{attribute 'linkalways'} 
{attribute 'no_explicit_call' := 'This FB is a CLASS and must be accessed using methods or properties'}
{attribute 'enable_dynamic_creation'}
FUNCTION_BLOCK Mc2Axis IMPLEMENTS Axis
VAR
	axis_ref : Tc2_Mc2.Axis_Ref;
	power_fb : Tc2_Mc2.Mc_Power;
	reset_fb : Tc2_Mc2.Mc_Reset;
	halt_fb : Tc2_Mc2.Mc_Halt;
	stop_fb : Tc2_Mc2.Mc_Stop;
END_VAR

METHOD PUBLIC CyclicCall
power_fb(Axis := axis_ref);
reset_fb(Axis := axis_ref);
halt_fb(Axis := axis_ref);
stop_fb(Axis := axis_ref);
axis_ref.ReadStatus();
END_METHOD

METHOD PUBLIC Disable
power_fb.Enable := FALSE;
power_fb.Enable_Positive := FALSE;
power_fb.Enable_Negative := FALSE;
END_METHOD

METHOD PUBLIC DisableNegative
power_fb.Enable_Negative := FALSE;
END_METHOD

METHOD PUBLIC DisablePositive
power_fb.Enable_Positive := FALSE;
END_METHOD

METHOD PUBLIC Enable
power_fb.Enable := TRUE;
END_METHOD

METHOD PUBLIC EnableNegative
power_fb.Enable_Negative := TRUE;
END_METHOD

METHOD PUBLIC EnablePositive
power_fb.Enable_Positive := TRUE;
END_METHOD

{attribute 'monitoring' := 'call'}
PROPERTY PUBLIC ErrorId : UDINT
GET // PUBLIC
ErrorId := axis_ref.Status.ErrorId;
END_GET
END_PROPERTY

METHOD PUBLIC GearIn : AsyncCommand
VAR_INPUT
	master_axis : Axis;
	numerator : LREAL;
	denominator : UINT := 1;
	//acceleration : LREAL := 0;
	//deceleration : LREAL := 0;
	//jerk : LREAL := 0;
	//buffer_mode	: MotionBufferMode := MotionBufferMode.Aborting;
END_VAR
VAR
	mc2_master_axis : POINTER TO Mc2Axis;
	command_pointer : POINTER TO GearInCommand;
END_VAR
IF __QUERYPOINTER(master_axis, mc2_master_axis) THEN
	command_pointer := __NEW(
		GearInCommand(
			master_axis := mc2_master_axis^,
			slave_axis := THIS^,
			numerator := numerator,
			denominator := denominator
		)
	);
	
	GearIn := command_pointer^;
END_IF
END_METHOD

METHOD PUBLIC GearOut : AsyncCommand
VAR
	command_pointer : POINTER TO GearOutCommand;
END_VAR
command_pointer := __NEW(
	GearOutCommand(
		axis := THIS^
	)
);

GearOut := command_pointer^;
END_METHOD

METHOD PUBLIC Halt : MoveCommand
VAR_INPUT
	deceleration : LREAL := 0;
	jerk : LREAL := 0;
	buffer_mode	: MotionBufferMode := MotionBufferMode.Aborting;
END_VAR
VAR
	command_pointer : POINTER TO HaltCommand;
END_VAR
command_pointer := __NEW(
	HaltCommand(
		axis := THIS^,
		deceleration := deceleration,
		jerk := jerk,
		buffer_mode := buffer_mode
	)
);

Halt := command_pointer^;
END_METHOD

{attribute 'monitoring' := 'call'}
PROPERTY PUBLIC HasBeenStopped : BOOL
GET // PUBLIC
HasBeenStopped := axis_ref.Status.HasBeenStopped;
END_GET
END_PROPERTY

{attribute 'monitoring' := 'call'}
PROPERTY PUBLIC HasJob : BOOL
GET // PUBLIC
HasJob := axis_ref.Status.HasJob;
END_GET
END_PROPERTY

{attribute 'monitoring' := 'call'}
PROPERTY PUBLIC IsAccelerating : BOOL
GET // PUBLIC
IsAccelerating := axis_ref.Status.Accelerating;
END_GET
END_PROPERTY

{attribute 'monitoring' := 'call'}
PROPERTY PUBLIC IsBusyHoming : BOOL
GET // PUBLIC
IsBusyHoming := axis_ref.Status.HomingBusy;
END_GET
END_PROPERTY

{attribute 'monitoring' := 'call'}
PROPERTY PUBLIC IsCamDataQueued : BOOL
GET // PUBLIC
IsCamDataQueued := axis_ref.Status.CamDataQueued;
END_GET
END_PROPERTY

{attribute 'monitoring' := 'call'}
PROPERTY PUBLIC IsCamScalingPending : BOOL
GET // PUBLIC
IsCamScalingPending := axis_ref.Status.CamScalingPending;
END_GET
END_PROPERTY

{attribute 'monitoring' := 'call'}
PROPERTY PUBLIC IsCamTableQueued : BOOL
GET // PUBLIC
IsCamTableQueued := axis_ref.Status.CamTableQueued;
END_GET
END_PROPERTY

{attribute 'monitoring' := 'call'}
 PROPERTY PUBLIC IsCommandBuffered : BOOL
GET // PUBLIC
IsCommandBuffered := axis_ref.Status.CmdBuffered;
END_GET
END_PROPERTY

{attribute 'monitoring' := 'call'}
PROPERTY PUBLIC IsCompensating : BOOL
GET // PUBLIC
IsCompensating := axis_ref.Status.Compensating;
END_GET
END_PROPERTY

{attribute 'monitoring' := 'call'}
PROPERTY PUBLIC IsConstantVelocity : BOOL
GET // PUBLIC
IsConstantVelocity := axis_ref.Status.ConstantVelocity;
END_GET
END_PROPERTY

{attribute 'monitoring' := 'call'}
PROPERTY PUBLIC IsContinuousMotion : BOOL
GET // PUBLIC
IsContinuousMotion := axis_ref.Status.ContinuousMotion;
END_GET
END_PROPERTY

{attribute 'monitoring' := 'call'}
PROPERTY PUBLIC IsControlLoopClosed : BOOL
GET // PUBLIC
IsControlLoopClosed := axis_ref.Status.ControlLoopClosed;
END_GET
END_PROPERTY

{attribute 'monitoring' := 'call'}
PROPERTY PUBLIC IsCoupled : BOOL
GET // PUBLIC
IsCoupled := axis_ref.Status.Coupled;
END_GET
END_PROPERTY

{attribute 'monitoring' := 'call'}
PROPERTY PUBLIC IsDecelerating : BOOL
GET // PUBLIC
IsDecelerating := axis_ref.Status.Decelerating;
END_GET
END_PROPERTY

{attribute 'monitoring' := 'call'}
PROPERTY PUBLIC IsDisabled : BOOL
GET // PUBLIC
IsDisabled := axis_ref.Status.Disabled;
END_GET
END_PROPERTY

{attribute 'monitoring' := 'call'}
PROPERTY PUBLIC IsDiscreteMotion : BOOL
GET // PUBLIC
END_GET
END_PROPERTY

{attribute 'monitoring' := 'call'}
PROPERTY PUBLIC IsDriveDeviceErrored : BOOL
GET // PUBLIC
IsDriveDeviceErrored := axis_ref.Status.Error;
END_GET
END_PROPERTY

{attribute 'monitoring' := 'call'}
PROPERTY PUBLIC IsErrored : BOOL
GET // PUBLIC
IsErrored := axis_ref.Status.Error;
END_GET
END_PROPERTY

{attribute 'monitoring' := 'call'}
PROPERTY PUBLIC IsErrorStop : BOOL
GET // PUBLIC
IsErrorStop := axis_ref.Status.ErrorStop;
END_GET
END_PROPERTY

{attribute 'monitoring' := 'call'}
PROPERTY PUBLIC IsExternalLatchValid : BOOL
GET // PUBLIC
IsExternalLatchValid := axis_ref.Status.ExternalLatchValid;
END_GET
END_PROPERTY

{attribute 'monitoring' := 'call'}
PROPERTY PUBLIC IsExtSetPointGenEnabled : BOOL
GET // PUBLIC
IsExtSetPointGenEnabled := axis_ref.Status.ExtSetPointGenEnabled;
END_GET
END_PROPERTY

{attribute 'monitoring' := 'call'}
PROPERTY PUBLIC IsHomed : BOOL
GET // PUBLIC
IsHomed := axis_ref.Status.Homed;
END_GET
END_PROPERTY

{attribute 'monitoring' := 'call'}
PROPERTY PUBLIC IsHoming : BOOL
GET // PUBLIC
IsHoming := axis_ref.Status.Homing;
END_GET
END_PROPERTY

{attribute 'monitoring' := 'call'}
PROPERTY PUBLIC IsInPositionArea : BOOL
GET // PUBLIC
IsInPositionArea := axis_ref.Status.InPositionArea;
END_GET
END_PROPERTY

{attribute 'monitoring' := 'call'}
PROPERTY PUBLIC IsInTargetPosition : BOOL
GET // PUBLIC
IsInTargetPosition := axis_ref.Status.InTargetPosition;
END_GET
END_PROPERTY

{attribute 'monitoring' := 'call'}
PROPERTY PUBLIC IsIoDataInvalid : BOOL
GET // PUBLIC
IsIoDataInvalid := axis_ref.Status.IoDataInvalid;
END_GET
END_PROPERTY

{attribute 'monitoring' := 'call'}
PROPERTY PUBLIC IsMotionCommandsLocked : BOOL
GET // PUBLIC
IsMotionCommandsLocked := axis_ref.Status.MotionCommandsLocked;
END_GET
END_PROPERTY

{attribute 'monitoring' := 'call'}
PROPERTY PUBLIC IsMoving : BOOL
GET // PUBLIC
IsMoving := axis_ref.Status.Moving;
END_GET
END_PROPERTY

{attribute 'monitoring' := 'call'}
PROPERTY PUBLIC IsNegativeDirection : BOOL
GET // PUBLIC
IsNegativeDirection := axis_ref.Status.NegativeDirection;
END_GET
END_PROPERTY

{attribute 'monitoring' := 'call'}
PROPERTY PUBLIC IsNewTargetPosition : BOOL
GET // PUBLIC
IsNewTargetPosition := axis_ref.Status.NewTargetPosition;
END_GET
END_PROPERTY

{attribute 'monitoring' := 'call'}
PROPERTY PUBLIC IsNotMoving : BOOL
GET // PUBLIC
IsNotMoving := axis_ref.Status.NotMoving;
END_GET
END_PROPERTY

{attribute 'monitoring' := 'call'}
PROPERTY PUBLIC IsOperational : BOOL
GET // PUBLIC
IsOperational := axis_ref.Status.Operational;
END_GET
END_PROPERTY

{attribute 'monitoring' := 'call'}
PROPERTY PUBLIC IsPointToPointMode : BOOL
GET // PUBLIC
IsPointToPointMode := axis_ref.Status.PTPmode;
END_GET
END_PROPERTY

{attribute 'monitoring' := 'call'}
PROPERTY PUBLIC IsPositiveDirection : BOOL
GET // PUBLIC
IsPositiveDirection := axis_ref.Status.PositiveDirection;
END_GET
END_PROPERTY

{attribute 'monitoring' := 'call'}
PROPERTY PUBLIC IsProtected : BOOL
GET // PUBLIC
IsProtected := axis_ref.Status.ProtectedMode;
END_GET
END_PROPERTY

{attribute 'monitoring' := 'call'}
PROPERTY PUBLIC IsSoftLimitMaxExceeded : BOOL
GET // PUBLIC
IsSoftLimitMaxExceeded := axis_ref.Status.SoftLimitMaxExceeded;
END_GET
END_PROPERTY

{attribute 'monitoring' := 'call'}
PROPERTY PUBLIC IsSoftLimitMinExceeded : BOOL
GET // PUBLIC
IsSoftLimitMinExceeded := axis_ref.Status.SoftLimitMinExceeded;
END_GET
END_PROPERTY

{attribute 'monitoring' := 'call'}
PROPERTY PUBLIC IsStandstill : BOOL
GET // PUBLIC
IsStandstill := axis_ref.Status.StandStill;
END_GET
END_PROPERTY

{attribute 'monitoring' := 'call'}
PROPERTY PUBLIC IsStopping : BOOL
GET // PUBLIC
IsStopping := axis_ref.Status.Stopping;
END_GET
END_PROPERTY

{attribute 'monitoring' := 'call'}
PROPERTY PUBLIC IsSynchronisedMotion : BOOL
GET // PUBLIC
IsSynchronisedMotion := axis_ref.Status.SynchronizedMotion;
END_GET
END_PROPERTY

PROPERTY PUBLIC Mc2AxisRef : REFERENCE TO Tc2_Mc2.Axis_Ref
GET // PUBLIC
Mc2AxisRef REF= THIS^.axis_ref;
END_GET
END_PROPERTY

{attribute 'monitoring' := 'call'}
PROPERTY PUBLIC MotionState : AxisMotionState
GET // PUBLIC
CASE axis_ref.Status.MotionState OF
	Tc2_Mc2.Mc_AxisState_Disabled: MotionState := AxisMotionState.Disabled;
	Tc2_Mc2.Mc_AxisState_Standstill: MotionState := AxisMotionState.Standstill;
	Tc2_Mc2.Mc_AxisState_ErrorStop: MotionState := AxisMotionState.ErrorStop;
	Tc2_Mc2.Mc_AxisState_Stopping: MotionState := AxisMotionState.Stopping;
	Tc2_Mc2.Mc_AxisState_Homing: MotionState := AxisMotionState.Homing;
	Tc2_Mc2.Mc_AxisState_DiscreteMotion: MotionState := AxisMotionState.DiscreteMotion;
	Tc2_Mc2.Mc_AxisState_ContinousMotion: MotionState := AxisMotionState.ContinuousMotion;
	Tc2_Mc2.Mc_AxisState_SynchronizedMotion: MotionState := AxisMotionState.SynchronisedMotion;
ELSE
	MotionState := AxisMotionState.Undefined;
END_CASE
END_GET
END_PROPERTY

METHOD PUBLIC MoveAbsolute : MoveCommand
VAR_INPUT
	position : LREAL;
	velocity : LREAL;
	acceleration : LREAL := 0;
	deceleration : LREAL := 0;
	jerk : LREAL := 0;
	buffer_mode	: MotionBufferMode := MotionBufferMode.Aborting;
END_VAR
VAR
	command_pointer : POINTER TO MoveAbsoluteCommand;
END_VAR
command_pointer := __NEW(
	MoveAbsoluteCommand(
		axis := THIS^,
		position := position,
		velocity := velocity,
		acceleration := acceleration,
		deceleration := deceleration,
		jerk := jerk,
		buffer_mode := buffer_mode
	)
);

MoveAbsolute := command_pointer^;
END_METHOD

METHOD PUBLIC MoveContinuousAbsolute : MoveCommand
VAR_INPUT
	position : LREAL;
	velocity : LREAL;
	acceleration : LREAL := 0;
	deceleration : LREAL := 0;
	jerk : LREAL := 0;
	buffer_mode	: MotionBufferMode := MotionBufferMode.Aborting;
END_VAR
VAR
	command_pointer : POINTER TO MoveContinuousAbsoluteCommand;
END_VAR
command_pointer := __NEW(
	MoveContinuousAbsoluteCommand(
		axis := THIS^,
		position := position,
		velocity := velocity,
		acceleration := acceleration,
		deceleration := deceleration,
		jerk := jerk,
		buffer_mode := buffer_mode
	)
);

MoveContinuousAbsolute := command_pointer^;
END_METHOD

METHOD PUBLIC MoveContinuousRelative : MoveCommand
VAR_INPUT
	distance : LREAL;
	velocity : LREAL;
	acceleration : LREAL := 0;
	deceleration : LREAL := 0;
	jerk : LREAL := 0;
	buffer_mode	: MotionBufferMode := MotionBufferMode.Aborting;
END_VAR
VAR
	command_pointer : POINTER TO MoveContinuousRelativeCommand;
END_VAR
command_pointer := __NEW(
	MoveContinuousRelativeCommand(
		axis := THIS^,
		distance := distance,
		velocity := velocity,
		acceleration := acceleration,
		deceleration := deceleration,
		jerk := jerk,
		buffer_mode := buffer_mode
	)
);

MoveContinuousRelative := command_pointer^;
END_METHOD

METHOD PUBLIC MoveModulo : MoveCommand
VAR_INPUT
	position : LREAL;
	direction : MotionDirection;
	velocity : LREAL;
	acceleration : LREAL := 0;
	deceleration : LREAL := 0;
	jerk : LREAL := 0;
	buffer_mode	: MotionBufferMode := MotionBufferMode.Aborting;
END_VAR
VAR
	command_pointer : POINTER TO MoveModuloCommand;
END_VAR
command_pointer := __NEW(
	MoveModuloCommand(
		axis := THIS^,
		position := position,
		direction := direction,
		velocity := velocity,
		acceleration := acceleration,
		deceleration := deceleration,
		jerk := jerk,
		buffer_mode := buffer_mode
	)
);

MoveModulo := command_pointer^;
END_METHOD

METHOD PUBLIC MoveRelative : MoveCommand
VAR_INPUT
	distance : LREAL;
	velocity : LREAL;
	acceleration : LREAL := 0;
	deceleration : LREAL := 0;
	jerk : LREAL := 0;
	buffer_mode	: MotionBufferMode := MotionBufferMode.Aborting;
END_VAR
VAR
	command_pointer : POINTER TO MoveRelativeCommand;
END_VAR
command_pointer := __NEW(
	MoveRelativeCommand(
		axis := THIS^,
		distance := distance,
		velocity := velocity,
		acceleration := acceleration,
		deceleration := deceleration,
		jerk := jerk,
		buffer_mode := buffer_mode
	)
);

MoveRelative := command_pointer^;
END_METHOD

METHOD PUBLIC MoveVelocity : MoveCommand
VAR_INPUT
	velocity : LREAL;
	acceleration : LREAL := 0;
	deceleration : LREAL := 0;
	jerk : LREAL := 0;
	buffer_mode	: MotionBufferMode := MotionBufferMode.Aborting;
END_VAR
VAR
	command_pointer : POINTER TO MoveVelocityCommand;
END_VAR
command_pointer := __NEW(
	MoveVelocityCommand(
		axis := THIS^,
		velocity := velocity,
		acceleration := acceleration,
		deceleration := deceleration,
		jerk := jerk,
		buffer_mode := buffer_mode
	)
);

MoveVelocity := command_pointer^;
END_METHOD

PROPERTY PUBLIC OpMode : Tc2_Mc2.St_AxisOpModes
GET // PUBLIC
OpMode := axis_ref.Status.OpMode;
END_GET
END_PROPERTY

METHOD PUBLIC Stop : MoveCommand
VAR_INPUT
	deceleration : LREAL := 0;
	jerk : LREAL := 0;
END_VAR
VAR
	command_pointer : POINTER TO StopCommand;
END_VAR
command_pointer := __NEW(
	StopCommand(
		axis := THIS^,
		deceleration := deceleration,
		jerk := jerk
	)
);

Stop := command_pointer^;
END_METHOD

END_FUNCTION_BLOCK

(* stored: Version 1.1.0.1
   POU Mc2Axis: Id {f6d24d44-bf88-05ab-17dd-e51bfbadd54a}, SpecialFunc None
   Folder Administrative: Id {c7a39c65-0d79-0e29-1377-7896a907f259}
   Folder Cyclic: Id {4bf04a9e-5f39-0347-2cc3-7f566b01be46}
   Folder Motion: Id {042d880c-d6a7-0bf4-26fc-fbf1514355b4}
   Folder Coupling: Id {c0c3d91b-c064-008c-3bc5-b7d09afefae3}
   Folder PointToPoint: Id {f7c42b14-1338-020f-0e42-fbe1e01f13ed}
   Folder Properties: Id {14bd5cf8-6829-0857-0543-912990d6f17c}
   Folder Error: Id {2ffa55bd-1a34-0c90-1876-f6f0946a309e}
   Folder States: Id {06982f99-509a-0977-0c86-36e4c9e4d884}
   Method CyclicCall: Id {c3d150dc-498f-087b-1e2a-cb28255a9a2e}
   Method Disable: Id {4475c6cd-2c80-0d86-32a6-2a6f85fa4e57}
   Method DisableNegative: Id {ab9e5fd9-cc11-0564-18aa-e34304f4e2e1}
   Method DisablePositive: Id {a7b584fc-cefd-0b94-3aad-fa7d09eaf38c}
   Method Enable: Id {51a4f218-30db-0a36-1b4f-54113e679d4a}
   Method EnableNegative: Id {1b82506a-a2bc-0e96-166c-a270fe33b5e2}
   Method EnablePositive: Id {5bc6496b-cc67-0922-28fc-331c9ad48fe1}
   Property ErrorId: Id {78f66620-fc8b-04ba-2c81-52c0f1fef6cb}
   Get Get: Id {572858b0-3000-039e-294f-09db91a746f0}
   Method GearIn: Id {19d44698-3c91-0578-1b51-8d7bddf03ae4}
   Method GearOut: Id {9f828a07-ad5e-0a29-08a3-d170a741d665}
   Method Halt: Id {bd9a8884-e367-05ac-2011-44121e4bfe1a}
   Property HasBeenStopped: Id {5da5e438-a929-084d-1690-b4c7d430baa3}
   Get Get: Id {05db3da7-bc46-0833-1b83-d37a59337621}
   Property HasJob: Id {523d496b-9657-07d6-055e-41f49b8ff99e}
   Get Get: Id {c3ce1acb-5d1c-0428-06e4-a53819984a3e}
   Property IsAccelerating: Id {ef93bcd0-2e43-098c-1e45-93ea63d85c21}
   Get Get: Id {3748b6f5-bad3-03a0-00b8-5541692d4281}
   Property IsBusyHoming: Id {78e0242c-43f6-00dd-1c0b-3a112bedd1f3}
   Get Get: Id {26cefb18-7e13-0f7c-3fd5-9a2d9a945033}
   Property IsCamDataQueued: Id {bfa5e2c6-a1b8-072e-1343-f2c82e2465be}
   Get Get: Id {0b42bbbc-7152-0758-1356-6a1b6ab20d4c}
   Property IsCamScalingPending: Id {de860177-b0c1-0299-154b-3806a6cdca90}
   Get Get: Id {766aa1a8-0d4f-0a15-39e4-a4660b05a7ae}
   Property IsCamTableQueued: Id {75ed77cd-a788-0e3f-31e7-de98fdd30099}
   Get Get: Id {d7ca3a57-bd1e-0e46-35f4-470c422ef820}
   Property IsCommandBuffered: Id {b037e227-a8b9-0e70-281b-08080b252061}
   Get Get: Id {8a4994b4-3b18-006c-3fb6-5613e0d8d1ee}
   Property IsCompensating: Id {316b11c2-e12a-069f-0be2-e4005b9003d4}
   Get Get: Id {fbc2ddf1-0a8a-0035-3b7a-a7896e19c528}
   Property IsConstantVelocity: Id {6a4d0ff6-a626-0141-307e-e4fe966b6439}
   Get Get: Id {8d2e3362-7b09-0633-0b5c-d5df8abd82b4}
   Property IsContinuousMotion: Id {9f4ef97f-2075-0ac0-350c-4a0af1ec6345}
   Get Get: Id {8ab7cb67-9d1e-0111-03e1-3647dd557e65}
   Property IsControlLoopClosed: Id {486a5c27-9a7c-0132-2b3d-22502f8b0d89}
   Get Get: Id {2062416c-cf8c-08bc-344f-0ef2f454f4b4}
   Property IsCoupled: Id {0e90c18b-5f7e-097f-1af7-f4b40426fa87}
   Get Get: Id {482e08a2-b9fb-0005-3233-477b456b0cbc}
   Property IsDecelerating: Id {5afc1dd6-c5b1-023c-2124-55b5060fb994}
   Get Get: Id {65bd9ee6-64dd-05fd-1de9-d2cfe2928e77}
   Property IsDisabled: Id {f757a26e-d51f-0b87-3f2a-165df82210b7}
   Get Get: Id {360a4cab-ee53-0d36-1188-4ca485d88d9c}
   Property IsDiscreteMotion: Id {6128acf7-fffa-0b89-0bd3-268f2e3ef87f}
   Get Get: Id {a134065a-97d7-092e-1f91-aec42a5fe214}
   Property IsDriveDeviceErrored: Id {8fba9b9f-e00b-0afa-1a40-033c77c15f6d}
   Get Get: Id {530d8c63-b6fb-0efc-1067-106ef31a8d19}
   Property IsErrored: Id {fb79de2a-70de-03ce-20b3-7e182dc76677}
   Get Get: Id {65d19f8f-3395-00d8-33df-359ddb0050db}
   Property IsErrorStop: Id {c23cd7da-639f-056e-354b-bedd34cd525b}
   Get Get: Id {ae835b87-db68-0f59-1fbb-a992e82263fd}
   Property IsExternalLatchValid: Id {379a565b-82b4-0d23-3b42-ba0e8e9de69c}
   Get Get: Id {227f0c80-7f76-0083-20f4-8fef89af8090}
   Property IsExtSetPointGenEnabled: Id {bf17920a-9b33-0c32-2dbd-9f7dd2872eb4}
   Get Get: Id {1c5b6205-c17d-05b0-0f8c-a8d2872fd975}
   Property IsHomed: Id {8a697d40-9c5a-0ddc-0c77-007dbc5d6060}
   Get Get: Id {1c2d286b-bf77-0fdc-0c67-ce0132c4b88f}
   Property IsHoming: Id {3d3a9cd9-3c28-00d2-23cd-3ffaae3f4dc8}
   Get Get: Id {3cbdd7b0-3538-0993-215f-c98e09cdfb99}
   Property IsInPositionArea: Id {d7721505-775c-0972-1a9c-d04ad8f80693}
   Get Get: Id {9c28b412-d198-0ccb-2b73-a4ffd412110e}
   Property IsInTargetPosition: Id {8a037e9a-6014-0f20-014c-1cb37ffabe8e}
   Get Get: Id {73be103e-8a2d-0202-2f33-617acbbc95f7}
   Property IsIoDataInvalid: Id {e586fbb9-881b-00a7-21a4-491863630ad3}
   Get Get: Id {44329c13-b919-09d5-24c1-55826d1d928c}
   Property IsMotionCommandsLocked: Id {8792db0e-b6e1-09bf-2a09-7eed78f99c4b}
   Get Get: Id {c93c0bfa-33c3-0178-2ce1-752ce0d58edb}
   Property IsMoving: Id {f0c8dcb7-c3ef-0a5a-2bfd-70089708db86}
   Get Get: Id {8bedff62-0000-0e2b-2c61-a40aa2e8e092}
   Property IsNegativeDirection: Id {1d0bbd0a-e60d-0563-2931-92b64cc23cd7}
   Get Get: Id {18e961b8-071d-05a5-3c48-d8569ec5fe58}
   Property IsNewTargetPosition: Id {f30cfb4b-9007-00dd-23ce-5428c054c856}
   Get Get: Id {be835f59-7610-05d4-046b-bbdc556e8eac}
   Property IsNotMoving: Id {40fe11d1-5990-0b21-399d-566f4ae6ffa3}
   Get Get: Id {9d66c255-2e58-08c5-16a8-21a9a8ec0f4a}
   Property IsOperational: Id {b4f3b1f9-9f4e-0b26-22d0-5b879ad50af2}
   Get Get: Id {28570211-377c-03fe-3da4-0c0537a51626}
   Property IsPointToPointMode: Id {8e61ad4d-3e20-0b40-0400-450a88f36809}
   Get Get: Id {e72289f6-b5dd-0b57-2378-44bddb740173}
   Property IsPositiveDirection: Id {3d940cdb-6245-0bf7-12c5-426feaf2df04}
   Get Get: Id {a0c27ab4-7afe-00f0-2938-2c9cbb9c1197}
   Property IsProtected: Id {f1d9e2db-1136-000e-2d22-dac81ddfd437}
   Get Get: Id {0f7f9efa-c917-0056-07e9-3ff374231520}
   Property IsSoftLimitMaxExceeded: Id {e914973f-eb5c-040b-3d6a-623c5105ea01}
   Get Get: Id {aca6918b-241a-0d01-1264-9caba7e27cce}
   Property IsSoftLimitMinExceeded: Id {172367ef-f52f-0fd1-1f93-f115f3ddf06e}
   Get Get: Id {86e3479c-522a-0d6a-2ed4-69925a8b156d}
   Property IsStandstill: Id {9cd772b9-621b-0d81-0ee2-1a0d2bdb6ebd}
   Get Get: Id {c5a99af5-a4bf-024d-0c88-bc9c19c4dc96}
   Property IsStopping: Id {ec574189-c78a-0dfb-29c3-2b0dfb259bf5}
   Get Get: Id {0b392166-cd5c-040e-2a41-3dc0ea9840a5}
   Property IsSynchronisedMotion: Id {e3ebe054-e597-0ab2-324d-e16e7f5d7836}
   Get Get: Id {94169aa8-2ebb-0267-2eda-e2ca94088856}
   Property Mc2AxisRef: Id {ae5866bb-3683-0a90-2259-7ccc10947c6c}
   Get Get: Id {fb8a0f8d-990d-0f9e-3f0c-06d665d956b7}
   Property MotionState: Id {c0cc5701-fbfb-05ed-3d3e-2b4764faf07c}
   Get Get: Id {b95dbae7-b719-0a18-321d-00327a4e6720}
   Method MoveAbsolute: Id {ba7aac53-f182-0124-2760-6e9ca44693a7}
   Method MoveContinuousAbsolute: Id {5ddeacc5-a151-0e3f-08e1-27b2f63b62da}
   Method MoveContinuousRelative: Id {2522a323-0580-0b3c-0982-42121392ccfc}
   Method MoveModulo: Id {3f82f632-2d6e-0a6c-000e-b08d835c76d4}
   Method MoveRelative: Id {55b852ad-4981-0b09-365a-969af570766f}
   Method MoveVelocity: Id {411c70a5-a751-02d2-30fb-eae8e1e29394}
   Property OpMode: Id {847e6f11-c9a7-0d26-1f26-0dcdf9c3787c}
   Get Get: Id {0c360fe3-6c1d-0982-34c6-93b59a552721}
   Method Stop: Id {a905c6b0-65a3-0b2e-0f5f-bf9f5c9e621b} *)
